// TIA Portal V20 export
DATA_BLOCK "HmiInterface"   // DB204
// stored: Access Published, MemoryReserve 100, Namespace Unit1
   VAR
      AutoStartEnable { ExternalWritable := 'False'} : Bool;
      InitializeEnable { ExternalWritable := 'False'} : Bool;
      camDataBk : Array[1..41] of "LER_typeSoftCamInterface";
   END_VAR
   VAR RETAIN
      BA010 : "LER_typeCommunicationInterface";
      BA015 : "LER_typeCommunicationInterface";
   END_VAR
   VAR
      BA060 { S7_SetPoint := 'True'} : "LER_typeCommunicationInterface";
      BA040 { S7_SetPoint := 'True'} : "LER_typeCommunicationInterface";
      cmFFU { S7_SetPoint := 'True'} : "LER_typeLIU117Interface";
      allBrakeTest : "LER_typeBrakeTestUnitInterface";
      cmPowerMeter_PAC3220 { S7_SetPoint := 'True'} : "LER_typePAC3220Interface";
      cmHandyQRreadDM8700 { S7_SetPoint := 'True'} : "LER_typeDM8700Interface";
      DriveDiagConfig : Struct
         driveObjects : Array[0..41] of "LAF_typeDriveDiagConfig";
         torqueLoad : Array[0.._.LAF_DRV_DIAG_NO_DO] of "LER_typeServoTorqueCalConfigruation";
      END_STRUCT;
      DriveDiagInterfaceHmi : Struct
         diagStatus : "LAF_typeDriveDiagInterfaceHmi";
         torqueLoad { S7_SetPoint := 'True'} : Array[0.._.LAF_DRV_DIAG_NO_DO] of "LER_typeServoTorqueCalInterface";
      END_STRUCT;
      ProductData_DriveSub : Int;
   END_VAR
BEGIN
   // camDataBk[3] : cmCompensatorAxisX
   // camDataBk[4] : cmSepaFeedingRollerAxisB
   // camDataBk[5] : anodeMainPnP1AxisX
   // camDataBk[6] : anodeMainPnP2AxisX
   // camDataBk[7] : cathodeMainPnP1AxisX
   // camDataBk[8] : cathodeMainPnP2AxisX
   // camDataBk[9] : cathodeMainPnP1AxisY
   // camDataBk[10] : cathodeMainPnP1AxisZ
   // camDataBk[11] : anodeMainPnP1AxisY
   // camDataBk[12] : anodeMainPnP1AxisZ
   // camDataBk[13] : cathodeMainPnP2AxisZ
   // camDataBk[14] : anodeMainPnP2AxisZ
   // camDataBk[15] : anodeAlignTableAxisX
   // camDataBk[16] : anodeAlignTableAxisY1
   // camDataBk[17] : anodeAlignTableAxisY2
   // camDataBk[18] : cathodeAlignTableAxisU
   // camDataBk[19] : cathodeAlignTableAxisV
   // camDataBk[20] : cathodeAlignTableAxisW
   // camDataBk[21] : FinalRollerFrontAxisX
   // camDataBk[22] : FinalRollerRearAxisX
   // camDataBk[23] : mendrelAnodeFrontAxisY
   // camDataBk[24] : mendrelAnodeFrontAxisZ
   // camDataBk[25] : mendrelAnodeRearAxisY
   // camDataBk[26] : mendrelAnodeRearAxisZ
   // camDataBk[27] : mendrelCathodeFrontAxisY
   // camDataBk[28] : mendrelCathodeFrontAxisZ
   // camDataBk[29] : mendrelCathodeRearAxisY
   // camDataBk[30] : mendrelCathodeRearAxisZ
   // camDataBk[31] : StackTableAxisZ
   // camDataBk[32] : StackTableOutFrontAxisZ
   // camDataBk[33] : StackTableOutRearAxisZ
   // camDataBk[34] : SepaClampnCutterAxisX
   // camDataBk[35] : SepaClampnCutterAxisZ
   // camDataBk[36] : SepaGripperAxisX
   // camDataBk[37] : SepaGripperAxisZ
   // camDataBk[38] : SepaGripperAxisC
   // camDataBk[39] : JRWinderFrontAxisY
   // camDataBk[40] : JRWinderRearAxisY
   // camDataBk[41] : JRWinderAxisB
   camDataBk[1..4].TargetPosition := 0.0;
   camDataBk[5].TargetPosition := -5.0;
   camDataBk[6].TargetPosition := 546.5;
   camDataBk[7..9].TargetPosition := 0.0;
   camDataBk[10].TargetPosition := 26.2;
   camDataBk[11..12].TargetPosition := 0.0;
   camDataBk[13].TargetPosition := 4.0;
   camDataBk[14].TargetPosition := 3.0;
   camDataBk[15].TargetPosition := -2.08;
   camDataBk[16].TargetPosition := 0.0;
   camDataBk[17].TargetPosition := 8.5;
   camDataBk[18..22].TargetPosition := 0.0;
   camDataBk[23].TargetPosition := 87.68;
   camDataBk[24].TargetPosition := 13.6;
   camDataBk[25].TargetPosition := 8.54;
   camDataBk[26].TargetPosition := -0.1;
   camDataBk[27].TargetPosition := 10.05;
   camDataBk[28].TargetPosition := -0.2;
   camDataBk[29].TargetPosition := 12.45;
   camDataBk[30].TargetPosition := -0.6;
   camDataBk[31].TargetPosition := -20.2;
   camDataBk[32..35].TargetPosition := 0.0;
   camDataBk[36].TargetPosition := 27.5;
   camDataBk[37..38].TargetPosition := 0.0;
   camDataBk[39].TargetPosition := -22.0;
   camDataBk[40..41].TargetPosition := 0.0;
   camDataBk[1..3].ActualPosition := 0.0;
   camDataBk[4].ActualPosition := 70.013;
   camDataBk[5].ActualPosition := 539.942;
   camDataBk[6].ActualPosition := 546.453;
   camDataBk[7].ActualPosition := 0.048;
   camDataBk[8].ActualPosition := -11.987;
   camDataBk[9].ActualPosition := 0.0;
   camDataBk[10].ActualPosition := 4.235;
   camDataBk[11].ActualPosition := 0.0;
   camDataBk[12].ActualPosition := 5.435;
   camDataBk[13].ActualPosition := 4.649;
   camDataBk[14].ActualPosition := 3.012;
   camDataBk[15].ActualPosition := -2.08;
   camDataBk[16].ActualPosition := 0.6;
   camDataBk[17].ActualPosition := 0.0;
   camDataBk[18].ActualPosition := -0.929;
   camDataBk[19].ActualPosition := 0.15;
   camDataBk[20].ActualPosition := -0.959;
   camDataBk[21].ActualPosition := 31.141;
   camDataBk[22].ActualPosition := 0.0;
   camDataBk[23].ActualPosition := -25.432;
   camDataBk[24].ActualPosition := 20.924;
   camDataBk[25].ActualPosition := 8.538;
   camDataBk[26].ActualPosition := 13.346;
   camDataBk[27].ActualPosition := 10.959;
   camDataBk[28].ActualPosition := 2.036;
   camDataBk[29].ActualPosition := 12.418;
   camDataBk[30].ActualPosition := 13.294;
   camDataBk[31].ActualPosition := -20.2;
   camDataBk[32].ActualPosition := -13.254;
   camDataBk[33].ActualPosition := 0.0;
   camDataBk[34].ActualPosition := 245.002;
   camDataBk[35].ActualPosition := 144.852;
   camDataBk[36].ActualPosition := 27.536;
   camDataBk[37].ActualPosition := 158.76;
   camDataBk[38].ActualPosition := -6.304;
   camDataBk[39].ActualPosition := -21.985;
   camDataBk[40].ActualPosition := -17.994;
   camDataBk[41].ActualPosition := 0.34;
   camDataBk[1..41].error := FALSE;
   camDataBk[1..41].status := 16#0000;
   camDataBk[1].position[0..8].SetValue.Negative := 0.0;
   camDataBk[2].position[0..8].SetValue.Negative := 0.0;
   camDataBk[3].position[0..8].SetValue.Negative := 1.0;
   camDataBk[4].position[0].SetValue.Negative := 0.0;
   camDataBk[4].position[1..2].SetValue.Negative := 1.0;
   camDataBk[4].position[3..8].SetValue.Negative := 0.0;
   camDataBk[5].position[0..8].SetValue.Negative := 1.0;
   camDataBk[6].position[0..8].SetValue.Negative := 1.0;
   camDataBk[7].position[0..8].SetValue.Negative := 1.0;
   camDataBk[8].position[0..8].SetValue.Negative := 1.0;
   camDataBk[9].position[0..8].SetValue.Negative := 1.0;
   camDataBk[10].position[0..8].SetValue.Negative := 1.0;
   camDataBk[11].position[0..8].SetValue.Negative := 1.0;
   camDataBk[12].position[0..8].SetValue.Negative := 1.0;
   camDataBk[13].position[0..8].SetValue.Negative := 1.0;
   camDataBk[14].position[0..8].SetValue.Negative := 1.0;
   camDataBk[15].position[0..8].SetValue.Negative := 1.0;
   camDataBk[16].position[0..8].SetValue.Negative := 1.0;
   camDataBk[17].position[0..8].SetValue.Negative := 1.0;
   camDataBk[18].position[0..8].SetValue.Negative := 1.0;
   camDataBk[19].position[0..8].SetValue.Negative := 1.0;
   camDataBk[20].position[0..8].SetValue.Negative := 1.0;
   camDataBk[21].position[0..8].SetValue.Negative := 1.0;
   camDataBk[22].position[0..8].SetValue.Negative := 1.0;
   camDataBk[23].position[0..8].SetValue.Negative := 1.0;
   camDataBk[24].position[0..8].SetValue.Negative := 1.0;
   camDataBk[25].position[0..8].SetValue.Negative := 1.0;
   camDataBk[26].position[0..8].SetValue.Negative := 1.0;
   camDataBk[27].position[0..8].SetValue.Negative := 1.0;
   camDataBk[28].position[0..8].SetValue.Negative := 1.0;
   camDataBk[29].position[0..8].SetValue.Negative := 1.0;
   camDataBk[30].position[0..8].SetValue.Negative := 1.0;
   camDataBk[31].position[0..8].SetValue.Negative := 1.0;
   camDataBk[32].position[0..8].SetValue.Negative := 1.0;
   camDataBk[33].position[0..8].SetValue.Negative := 1.0;
   camDataBk[34].position[0..8].SetValue.Negative := 1.0;
   camDataBk[35].position[0..8].SetValue.Negative := 1.0;
   camDataBk[36].position[0..8].SetValue.Negative := 1.0;
   camDataBk[37].position[0..8].SetValue.Negative := 1.0;
   camDataBk[38].position[0..8].SetValue.Negative := 1.0;
   camDataBk[39].position[0..8].SetValue.Negative := 1.0;
   camDataBk[40].position[0..8].SetValue.Negative := 1.0;
   camDataBk[41].position[0..8].SetValue.Negative := 1.0;
   camDataBk[1].position[0..8].SetValue.Postive := 0.0;
   camDataBk[2].position[0..8].SetValue.Postive := 0.0;
   camDataBk[3].position[0..8].SetValue.Postive := 1.0;
   camDataBk[4].position[0].SetValue.Postive := 0.0;
   camDataBk[4].position[1..2].SetValue.Postive := 1.0;
   camDataBk[4].position[3..8].SetValue.Postive := 0.0;
   camDataBk[5].position[0..8].SetValue.Postive := 1.0;
   camDataBk[6].position[0..8].SetValue.Postive := 1.0;
   camDataBk[7].position[0..5].SetValue.Postive := 1.0;
   camDataBk[7].position[6].SetValue.Postive := 0.001;
   camDataBk[7].position[7..8].SetValue.Postive := 1.0;
   camDataBk[8].position[0..8].SetValue.Postive := 1.0;
   camDataBk[9].position[0..8].SetValue.Postive := 1.0;
   camDataBk[10].position[0..8].SetValue.Postive := 1.0;
   camDataBk[11].position[0..8].SetValue.Postive := 1.0;
   camDataBk[12].position[0..8].SetValue.Postive := 1.0;
   camDataBk[13].position[0..8].SetValue.Postive := 1.0;
   camDataBk[14].position[0..8].SetValue.Postive := 1.0;
   camDataBk[15].position[0..8].SetValue.Postive := 1.0;
   camDataBk[16].position[0..8].SetValue.Postive := 1.0;
   camDataBk[17].position[0..8].SetValue.Postive := 1.0;
   camDataBk[18].position[0..8].SetValue.Postive := 1.0;
   camDataBk[19].position[0..8].SetValue.Postive := 1.0;
   camDataBk[20].position[0..8].SetValue.Postive := 1.0;
   camDataBk[21].position[0..8].SetValue.Postive := 1.0;
   camDataBk[22].position[0..8].SetValue.Postive := 1.0;
   camDataBk[23].position[0..8].SetValue.Postive := 1.0;
   camDataBk[24].position[0..8].SetValue.Postive := 1.0;
   camDataBk[25].position[0..8].SetValue.Postive := 1.0;
   camDataBk[26].position[0..8].SetValue.Postive := 1.0;
   camDataBk[27].position[0..8].SetValue.Postive := 1.0;
   camDataBk[28].position[0..8].SetValue.Postive := 1.0;
   camDataBk[29].position[0..8].SetValue.Postive := 1.0;
   camDataBk[30].position[0..8].SetValue.Postive := 1.0;
   camDataBk[31].position[0..8].SetValue.Postive := 1.0;
   camDataBk[32].position[0..8].SetValue.Postive := 1.0;
   camDataBk[33].position[0..8].SetValue.Postive := 1.0;
   camDataBk[34].position[0..8].SetValue.Postive := 1.0;
   camDataBk[35].position[0..8].SetValue.Postive := 1.0;
   camDataBk[36].position[0..8].SetValue.Postive := 1.0;
   camDataBk[37].position[0..8].SetValue.Postive := 1.0;
   camDataBk[38].position[0..8].SetValue.Postive := 1.0;
   camDataBk[39].position[0..8].SetValue.Postive := 1.0;
   camDataBk[40].position[0..8].SetValue.Postive := 1.0;
   camDataBk[41].position[0..8].SetValue.Postive := 1.0;
   camDataBk[1].position[0..8].ProcessValue.Postive := 0.0;
   camDataBk[2].position[0..8].ProcessValue.Postive := 0.0;
   camDataBk[3].position[0..8].ProcessValue.Postive := 0.0;
   camDataBk[4].position[0].ProcessValue.Postive := 0.0;
   camDataBk[4].position[1..2].ProcessValue.Postive := 1.0;
   camDataBk[4].position[3..8].ProcessValue.Postive := 0.0;
   camDataBk[5].position[0..8].ProcessValue.Postive := 1.0;
   camDataBk[6].position[0..8].ProcessValue.Postive := 1.0;
   camDataBk[7].position[0..5].ProcessValue.Postive := 1.0;
   camDataBk[7].position[6].ProcessValue.Postive := 0.001;
   camDataBk[7].position[7..8].ProcessValue.Postive := 1.0;
   camDataBk[8].position[0..8].ProcessValue.Postive := 1.0;
   camDataBk[9].position[0..8].ProcessValue.Postive := 1.0;
   camDataBk[10].position[0..8].ProcessValue.Postive := 1.0;
   camDataBk[11].position[0..8].ProcessValue.Postive := 1.0;
   camDataBk[12].position[0..8].ProcessValue.Postive := 1.0;
   camDataBk[13].position[0..8].ProcessValue.Postive := 1.0;
   camDataBk[14].position[0..8].ProcessValue.Postive := 1.0;
   camDataBk[15].position[0..8].ProcessValue.Postive := 1.0;
   camDataBk[16].position[0..8].ProcessValue.Postive := 1.0;
   camDataBk[17].position[0..8].ProcessValue.Postive := 1.0;
   camDataBk[18].position[0..8].ProcessValue.Postive := 1.0;
   camDataBk[19].position[0..8].ProcessValue.Postive := 1.0;
   camDataBk[20].position[0..8].ProcessValue.Postive := 1.0;
   camDataBk[21].position[0..8].ProcessValue.Postive := 1.0;
   camDataBk[22].position[0..8].ProcessValue.Postive := 0.0;
   camDataBk[23].position[0..8].ProcessValue.Postive := 1.0;
   camDataBk[24].position[0..8].ProcessValue.Postive := 1.0;
   camDataBk[25].position[0..8].ProcessValue.Postive := 1.0;
   camDataBk[26].position[0..8].ProcessValue.Postive := 1.0;
   camDataBk[27].position[0..8].ProcessValue.Postive := 1.0;
   camDataBk[28].position[0..8].ProcessValue.Postive := 1.0;
   camDataBk[29].position[0..8].ProcessValue.Postive := 1.0;
   camDataBk[30].position[0..8].ProcessValue.Postive := 1.0;
   camDataBk[31].position[0..8].ProcessValue.Postive := 1.0;
   camDataBk[32].position[0..8].ProcessValue.Postive := 1.0;
   camDataBk[33].position[0..8].ProcessValue.Postive := 0.0;
   camDataBk[34].position[0..8].ProcessValue.Postive := 1.0;
   camDataBk[35].position[0..8].ProcessValue.Postive := 1.0;
   camDataBk[36].position[0..8].ProcessValue.Postive := 1.0;
   camDataBk[37].position[0..8].ProcessValue.Postive := 1.0;
   camDataBk[38].position[0..8].ProcessValue.Postive := 1.0;
   camDataBk[39].position[0..8].ProcessValue.Postive := 1.0;
   camDataBk[40].position[0..8].ProcessValue.Postive := 1.0;
   camDataBk[41].position[0..8].ProcessValue.Postive := 1.0;
   camDataBk[1].position[0..8].ProcessValue.Negative := 0.0;
   camDataBk[2].position[0..8].ProcessValue.Negative := 0.0;
   camDataBk[3].position[0..8].ProcessValue.Negative := 0.0;
   camDataBk[4].position[0].ProcessValue.Negative := 0.0;
   camDataBk[4].position[1..2].ProcessValue.Negative := 1.0;
   camDataBk[4].position[3..8].ProcessValue.Negative := 0.0;
   camDataBk[5].position[0..8].ProcessValue.Negative := 1.0;
   camDataBk[6].position[0..8].ProcessValue.Negative := 1.0;
   camDataBk[7].position[0..8].ProcessValue.Negative := 1.0;
   camDataBk[8].position[0..8].ProcessValue.Negative := 1.0;
   camDataBk[9].position[0..8].ProcessValue.Negative := 1.0;
   camDataBk[10].position[0..8].ProcessValue.Negative := 1.0;
   camDataBk[11].position[0..8].ProcessValue.Negative := 1.0;
   camDataBk[12].position[0..8].ProcessValue.Negative := 1.0;
   camDataBk[13].position[0..8].ProcessValue.Negative := 1.0;
   camDataBk[14].position[0..8].ProcessValue.Negative := 1.0;
   camDataBk[15].position[0..8].ProcessValue.Negative := 1.0;
   camDataBk[16].position[0..8].ProcessValue.Negative := 1.0;
   camDataBk[17].position[0..8].ProcessValue.Negative := 1.0;
   camDataBk[18].position[0..8].ProcessValue.Negative := 1.0;
   camDataBk[19].position[0..8].ProcessValue.Negative := 1.0;
   camDataBk[20].position[0..8].ProcessValue.Negative := 1.0;
   camDataBk[21].position[0..8].ProcessValue.Negative := 1.0;
   camDataBk[22].position[0..8].ProcessValue.Negative := 0.0;
   camDataBk[23].position[0..8].ProcessValue.Negative := 1.0;
   camDataBk[24].position[0..8].ProcessValue.Negative := 1.0;
   camDataBk[25].position[0..8].ProcessValue.Negative := 1.0;
   camDataBk[26].position[0..8].ProcessValue.Negative := 1.0;
   camDataBk[27].position[0..8].ProcessValue.Negative := 1.0;
   camDataBk[28].position[0..8].ProcessValue.Negative := 1.0;
   camDataBk[29].position[0..8].ProcessValue.Negative := 1.0;
   camDataBk[30].position[0..8].ProcessValue.Negative := 1.0;
   camDataBk[31].position[0..8].ProcessValue.Negative := 1.0;
   camDataBk[32].position[0..8].ProcessValue.Negative := 1.0;
   camDataBk[33].position[0..8].ProcessValue.Negative := 0.0;
   camDataBk[34].position[0..8].ProcessValue.Negative := 1.0;
   camDataBk[35].position[0..8].ProcessValue.Negative := 1.0;
   camDataBk[36].position[0..8].ProcessValue.Negative := 1.0;
   camDataBk[37].position[0..8].ProcessValue.Negative := 1.0;
   camDataBk[38].position[0..8].ProcessValue.Negative := 1.0;
   camDataBk[39].position[0..8].ProcessValue.Negative := 1.0;
   camDataBk[40].position[0..8].ProcessValue.Negative := 1.0;
   camDataBk[41].position[0..8].ProcessValue.Negative := 1.0;
   camDataBk[1].position[0..8].ProcessValue.SetPos := 0.0;
   camDataBk[2].position[0..8].ProcessValue.SetPos := 0.0;
   camDataBk[3].position[0..8].ProcessValue.SetPos := 0.0;
   camDataBk[4].position[0].ProcessValue.SetPos := 0.0;
   camDataBk[4].position[1].ProcessValue.SetPos := 50.0;
   camDataBk[4].position[2].ProcessValue.SetPos := 70.0;
   camDataBk[4].position[3..8].ProcessValue.SetPos := 0.0;
   camDataBk[5].position[0].ProcessValue.SetPos := 0.0;
   camDataBk[5].position[1].ProcessValue.SetPos := 540.0;
   camDataBk[5].position[2].ProcessValue.SetPos := -5.0;
   camDataBk[5].position[3..8].ProcessValue.SetPos := 0.0;
   camDataBk[6].position[0].ProcessValue.SetPos := 0.0;
   camDataBk[6].position[1].ProcessValue.SetPos := 546.5;
   camDataBk[6].position[2].ProcessValue.SetPos := -3.5;
   camDataBk[6].position[3..8].ProcessValue.SetPos := 0.0;
   camDataBk[7].position[0..1].ProcessValue.SetPos := 0.0;
   camDataBk[7].position[2].ProcessValue.SetPos := 544.0;
   camDataBk[7].position[3..8].ProcessValue.SetPos := 0.0;
   camDataBk[8].position[0].ProcessValue.SetPos := 0.0;
   camDataBk[8].position[1].ProcessValue.SetPos := -12.0;
   camDataBk[8].position[2].ProcessValue.SetPos := 538.0;
   camDataBk[8].position[3..8].ProcessValue.SetPos := 0.0;
   camDataBk[9].position[0..8].ProcessValue.SetPos := 0.0;
   camDataBk[10].position[0].ProcessValue.SetPos := 0.0;
   camDataBk[10].position[1].ProcessValue.SetPos := 0.3;
   camDataBk[10].position[2].ProcessValue.SetPos := 26.2;
   camDataBk[10].position[3..8].ProcessValue.SetPos := 0.0;
   camDataBk[11].position[0..8].ProcessValue.SetPos := 0.0;
   camDataBk[12].position[0..1].ProcessValue.SetPos := 4.0;
   camDataBk[12].position[2].ProcessValue.SetPos := 23.0;
   camDataBk[12].position[3].ProcessValue.SetPos := 26.3;
   camDataBk[12].position[4..8].ProcessValue.SetPos := 0.0;
   camDataBk[13].position[0].ProcessValue.SetPos := 0.0;
   camDataBk[13].position[1].ProcessValue.SetPos := 4.0;
   camDataBk[13].position[2].ProcessValue.SetPos := 26.6;
   camDataBk[13].position[3..8].ProcessValue.SetPos := 0.0;
   camDataBk[14].position[0].ProcessValue.SetPos := 0.0;
   camDataBk[14].position[1].ProcessValue.SetPos := 3.0;
   camDataBk[14].position[2].ProcessValue.SetPos := 25.5;
   camDataBk[14].position[3].ProcessValue.SetPos := 26.5;
   camDataBk[14].position[4..8].ProcessValue.SetPos := 0.0;
   camDataBk[15].position[0].ProcessValue.SetPos := 0.0;
   camDataBk[15].position[1].ProcessValue.SetPos := -2.08;
   camDataBk[15].position[2..3].ProcessValue.SetPos := -4.08;
   camDataBk[15].position[4].ProcessValue.SetPos := -2.08;
   camDataBk[15].position[5..7].ProcessValue.SetPos := -0.08;
   camDataBk[15].position[8].ProcessValue.SetPos := 6.42;
   camDataBk[16].position[0].ProcessValue.SetPos := 0.0;
   camDataBk[16].position[1..2].ProcessValue.SetPos := 0.6;
   camDataBk[16].position[3..5].ProcessValue.SetPos := 2.6;
   camDataBk[16].position[6].ProcessValue.SetPos := 0.6;
   camDataBk[16].position[7].ProcessValue.SetPos := -1.4;
   camDataBk[16].position[8].ProcessValue.SetPos := 9.1;
   camDataBk[17].position[0..7].ProcessValue.SetPos := 0.0;
   camDataBk[17].position[8].ProcessValue.SetPos := 8.5;
   camDataBk[18].position[0].ProcessValue.SetPos := 0.0;
   camDataBk[18].position[1].ProcessValue.SetPos := -0.93;
   camDataBk[18].position[2..3].ProcessValue.SetPos := 1.07;
   camDataBk[18].position[4].ProcessValue.SetPos := -0.93;
   camDataBk[18].position[5..7].ProcessValue.SetPos := -2.93;
   camDataBk[18].position[8].ProcessValue.SetPos := -0.93;
   camDataBk[19].position[0].ProcessValue.SetPos := 0.0;
   camDataBk[19].position[1..2].ProcessValue.SetPos := 0.15;
   camDataBk[19].position[3..5].ProcessValue.SetPos := 2.15;
   camDataBk[19].position[6].ProcessValue.SetPos := 0.15;
   camDataBk[19].position[7].ProcessValue.SetPos := -1.85;
   camDataBk[19].position[8].ProcessValue.SetPos := 0.15;
   camDataBk[20].position[0].ProcessValue.SetPos := 0.0;
   camDataBk[20].position[1..2].ProcessValue.SetPos := -0.96;
   camDataBk[20].position[3..5].ProcessValue.SetPos := -2.96;
   camDataBk[20].position[6].ProcessValue.SetPos := -0.96;
   camDataBk[20].position[7].ProcessValue.SetPos := 1.04;
   camDataBk[20].position[8].ProcessValue.SetPos := -0.96;
   camDataBk[21].position[0].ProcessValue.SetPos := 0.0;
   camDataBk[21].position[1].ProcessValue.SetPos := -1.0;
   camDataBk[21].position[2].ProcessValue.SetPos := 345.0;
   camDataBk[21].position[3..8].ProcessValue.SetPos := 0.0;
   camDataBk[22].position[0..8].ProcessValue.SetPos := 0.0;
   camDataBk[23].position[0].ProcessValue.SetPos := 0.0;
   camDataBk[23].position[1].ProcessValue.SetPos := 12.44;
   camDataBk[23].position[2].ProcessValue.SetPos := 87.68;
   camDataBk[23].position[3..8].ProcessValue.SetPos := 0.0;
   camDataBk[24].position[0].ProcessValue.SetPos := 0.0;
   camDataBk[24].position[1].ProcessValue.SetPos := -2.8;
   camDataBk[24].position[2].ProcessValue.SetPos := 13.6;
   camDataBk[24].position[3..8].ProcessValue.SetPos := 0.0;
   camDataBk[25].position[0].ProcessValue.SetPos := 0.0;
   camDataBk[25].position[1].ProcessValue.SetPos := 8.54;
   camDataBk[25].position[2].ProcessValue.SetPos := 84.03;
   camDataBk[25].position[3..8].ProcessValue.SetPos := 0.0;
   camDataBk[26].position[0].ProcessValue.SetPos := 0.0;
   camDataBk[26].position[1].ProcessValue.SetPos := -0.1;
   camDataBk[26].position[2].ProcessValue.SetPos := 15.7;
   camDataBk[26].position[3..8].ProcessValue.SetPos := 0.0;
   camDataBk[27].position[0].ProcessValue.SetPos := 0.0;
   camDataBk[27].position[1].ProcessValue.SetPos := 10.05;
   camDataBk[27].position[2].ProcessValue.SetPos := 85.43;
   camDataBk[27].position[3..8].ProcessValue.SetPos := 0.0;
   camDataBk[28].position[0].ProcessValue.SetPos := 0.0;
   camDataBk[28].position[1].ProcessValue.SetPos := -0.2;
   camDataBk[28].position[2].ProcessValue.SetPos := 14.4;
   camDataBk[28].position[3..8].ProcessValue.SetPos := 0.0;
   camDataBk[29].position[0].ProcessValue.SetPos := 0.0;
   camDataBk[29].position[1].ProcessValue.SetPos := 12.45;
   camDataBk[29].position[2].ProcessValue.SetPos := 88.92;
   camDataBk[29].position[3..8].ProcessValue.SetPos := 0.0;
   camDataBk[30].position[0].ProcessValue.SetPos := 0.0;
   camDataBk[30].position[1].ProcessValue.SetPos := -0.6;
   camDataBk[30].position[2].ProcessValue.SetPos := 14.6;
   camDataBk[30].position[3..8].ProcessValue.SetPos := 0.0;
   camDataBk[31].position[0].ProcessValue.SetPos := 0.0;
   camDataBk[31].position[1].ProcessValue.SetPos := -20.2;
   camDataBk[31].position[2].ProcessValue.SetPos := 0.0;
   camDataBk[31].position[3].ProcessValue.SetPos := -3.5;
   camDataBk[31].position[4..8].ProcessValue.SetPos := 0.0;
   camDataBk[32].position[0].ProcessValue.SetPos := 0.0;
   camDataBk[32].position[1].ProcessValue.SetPos := -10.76;
   camDataBk[32].position[2].ProcessValue.SetPos := 174.0;
   camDataBk[32].position[3..8].ProcessValue.SetPos := 0.0;
   camDataBk[33].position[0..8].ProcessValue.SetPos := 0.0;
   camDataBk[34].position[0].ProcessValue.SetPos := 0.0;
   camDataBk[34].position[1].ProcessValue.SetPos := 245.0;
   camDataBk[34].position[2].ProcessValue.SetPos := 48.2;
   camDataBk[34].position[3].ProcessValue.SetPos := 720.0;
   camDataBk[34].position[4..8].ProcessValue.SetPos := 0.0;
   camDataBk[35].position[0].ProcessValue.SetPos := 0.0;
   camDataBk[35].position[1].ProcessValue.SetPos := 141.0;
   camDataBk[35].position[2].ProcessValue.SetPos := 143.8;
   camDataBk[35].position[3].ProcessValue.SetPos := 160.0;
   camDataBk[35].position[4..8].ProcessValue.SetPos := 0.0;
   camDataBk[36].position[0].ProcessValue.SetPos := 0.0;
   camDataBk[36].position[1].ProcessValue.SetPos := 27.5;
   camDataBk[36].position[2..3].ProcessValue.SetPos := 1706.6;
   camDataBk[36].position[4].ProcessValue.SetPos := 245.0;
   camDataBk[36].position[5].ProcessValue.SetPos := 27.5;
   camDataBk[36].position[6].ProcessValue.SetPos := 227.5;
   camDataBk[36].position[7].ProcessValue.SetPos := 0.0;
   camDataBk[36].position[8].ProcessValue.SetPos := 179.3;
   camDataBk[37].position[0].ProcessValue.SetPos := 0.0;
   camDataBk[37].position[1].ProcessValue.SetPos := 233.0;
   camDataBk[37].position[2].ProcessValue.SetPos := 280.6;
   camDataBk[37].position[3].ProcessValue.SetPos := 159.6;
   camDataBk[37].position[4].ProcessValue.SetPos := 18.75;
   camDataBk[37].position[5].ProcessValue.SetPos := 233.5;
   camDataBk[37].position[6].ProcessValue.SetPos := 146.0;
   camDataBk[37].position[7..8].ProcessValue.SetPos := 0.0;
   camDataBk[38].position[0].ProcessValue.SetPos := 0.0;
   camDataBk[38].position[1].ProcessValue.SetPos := -1.43;
   camDataBk[38].position[2].ProcessValue.SetPos := 178.4;
   camDataBk[38].position[3].ProcessValue.SetPos := 88.4;
   camDataBk[38].position[4..8].ProcessValue.SetPos := 0.0;
   camDataBk[39].position[0].ProcessValue.SetPos := 0.0;
   camDataBk[39].position[1].ProcessValue.SetPos := -22.0;
   camDataBk[39].position[2].ProcessValue.SetPos := 160.0;
   camDataBk[39].position[3..8].ProcessValue.SetPos := 0.0;
   camDataBk[40].position[0].ProcessValue.SetPos := 0.0;
   camDataBk[40].position[1..2].ProcessValue.SetPos := -18.0;
   camDataBk[40].position[3..8].ProcessValue.SetPos := 0.0;
   camDataBk[41].position[0..8].ProcessValue.SetPos := 0.0;
   camDataBk[1].position[0..8].ProcessValue.inPos := FALSE;
   camDataBk[2].position[0..8].ProcessValue.inPos := FALSE;
   camDataBk[3].position[0..8].ProcessValue.inPos := FALSE;
   camDataBk[4].position[0..1].ProcessValue.inPos := FALSE;
   camDataBk[4].position[2].ProcessValue.inPos := TRUE;
   camDataBk[4].position[3..8].ProcessValue.inPos := FALSE;
   camDataBk[5].position[0].ProcessValue.inPos := FALSE;
   camDataBk[5].position[1].ProcessValue.inPos := TRUE;
   camDataBk[5].position[2..8].ProcessValue.inPos := FALSE;
   camDataBk[6].position[0].ProcessValue.inPos := FALSE;
   camDataBk[6].position[1].ProcessValue.inPos := TRUE;
   camDataBk[6].position[2..8].ProcessValue.inPos := FALSE;
   camDataBk[7].position[0..1].ProcessValue.inPos := TRUE;
   camDataBk[7].position[2].ProcessValue.inPos := FALSE;
   camDataBk[7].position[3..5].ProcessValue.inPos := TRUE;
   camDataBk[7].position[6].ProcessValue.inPos := FALSE;
   camDataBk[7].position[7..8].ProcessValue.inPos := TRUE;
   camDataBk[8].position[0].ProcessValue.inPos := FALSE;
   camDataBk[8].position[1].ProcessValue.inPos := TRUE;
   camDataBk[8].position[2..8].ProcessValue.inPos := FALSE;
   camDataBk[9].position[0..8].ProcessValue.inPos := TRUE;
   camDataBk[10].position[0..8].ProcessValue.inPos := FALSE;
   camDataBk[11].position[0..8].ProcessValue.inPos := TRUE;
   camDataBk[12].position[0..8].ProcessValue.inPos := FALSE;
   camDataBk[13].position[0].ProcessValue.inPos := FALSE;
   camDataBk[13].position[1].ProcessValue.inPos := TRUE;
   camDataBk[13].position[2..8].ProcessValue.inPos := FALSE;
   camDataBk[14].position[0].ProcessValue.inPos := FALSE;
   camDataBk[14].position[1].ProcessValue.inPos := TRUE;
   camDataBk[14].position[2..8].ProcessValue.inPos := FALSE;
   camDataBk[15].position[0].ProcessValue.inPos := FALSE;
   camDataBk[15].position[1].ProcessValue.inPos := TRUE;
   camDataBk[15].position[2..3].ProcessValue.inPos := FALSE;
   camDataBk[15].position[4].ProcessValue.inPos := TRUE;
   camDataBk[15].position[5..8].ProcessValue.inPos := FALSE;
   camDataBk[16].position[0..2].ProcessValue.inPos := TRUE;
   camDataBk[16].position[3..5].ProcessValue.inPos := FALSE;
   camDataBk[16].position[6].ProcessValue.inPos := TRUE;
   camDataBk[16].position[7..8].ProcessValue.inPos := FALSE;
   camDataBk[17].position[0..7].ProcessValue.inPos := TRUE;
   camDataBk[17].position[8].ProcessValue.inPos := FALSE;
   camDataBk[18].position[0..1].ProcessValue.inPos := TRUE;
   camDataBk[18].position[2..3].ProcessValue.inPos := FALSE;
   camDataBk[18].position[4].ProcessValue.inPos := TRUE;
   camDataBk[18].position[5..7].ProcessValue.inPos := FALSE;
   camDataBk[18].position[8].ProcessValue.inPos := TRUE;
   camDataBk[19].position[0..2].ProcessValue.inPos := TRUE;
   camDataBk[19].position[3..5].ProcessValue.inPos := FALSE;
   camDataBk[19].position[6].ProcessValue.inPos := TRUE;
   camDataBk[19].position[7].ProcessValue.inPos := FALSE;
   camDataBk[19].position[8].ProcessValue.inPos := TRUE;
   camDataBk[20].position[0..2].ProcessValue.inPos := TRUE;
   camDataBk[20].position[3..5].ProcessValue.inPos := FALSE;
   camDataBk[20].position[6].ProcessValue.inPos := TRUE;
   camDataBk[20].position[7].ProcessValue.inPos := FALSE;
   camDataBk[20].position[8].ProcessValue.inPos := TRUE;
   camDataBk[21].position[0..8].ProcessValue.inPos := FALSE;
   camDataBk[22].position[0..8].ProcessValue.inPos := FALSE;
   camDataBk[23].position[0..8].ProcessValue.inPos := FALSE;
   camDataBk[24].position[0..8].ProcessValue.inPos := FALSE;
   camDataBk[25].position[0].ProcessValue.inPos := FALSE;
   camDataBk[25].position[1].ProcessValue.inPos := TRUE;
   camDataBk[25].position[2..8].ProcessValue.inPos := FALSE;
   camDataBk[26].position[0..8].ProcessValue.inPos := FALSE;
   camDataBk[27].position[0].ProcessValue.inPos := FALSE;
   camDataBk[27].position[1].ProcessValue.inPos := TRUE;
   camDataBk[27].position[2..8].ProcessValue.inPos := FALSE;
   camDataBk[28].position[0..8].ProcessValue.inPos := FALSE;
   camDataBk[29].position[0].ProcessValue.inPos := FALSE;
   camDataBk[29].position[1].ProcessValue.inPos := TRUE;
   camDataBk[29].position[2..8].ProcessValue.inPos := FALSE;
   camDataBk[30].position[0..8].ProcessValue.inPos := FALSE;
   camDataBk[31].position[0].ProcessValue.inPos := FALSE;
   camDataBk[31].position[1].ProcessValue.inPos := TRUE;
   camDataBk[31].position[2..8].ProcessValue.inPos := FALSE;
   camDataBk[32].position[0..8].ProcessValue.inPos := FALSE;
   camDataBk[33].position[0..8].ProcessValue.inPos := FALSE;
   camDataBk[34].position[0].ProcessValue.inPos := FALSE;
   camDataBk[34].position[1].ProcessValue.inPos := TRUE;
   camDataBk[34].position[2..8].ProcessValue.inPos := FALSE;
   camDataBk[35].position[0..8].ProcessValue.inPos := FALSE;
   camDataBk[36].position[0].ProcessValue.inPos := FALSE;
   camDataBk[36].position[1].ProcessValue.inPos := TRUE;
   camDataBk[36].position[2..4].ProcessValue.inPos := FALSE;
   camDataBk[36].position[5].ProcessValue.inPos := TRUE;
   camDataBk[36].position[6..8].ProcessValue.inPos := FALSE;
   camDataBk[37].position[0..2].ProcessValue.inPos := FALSE;
   camDataBk[37].position[3].ProcessValue.inPos := TRUE;
   camDataBk[37].position[4..8].ProcessValue.inPos := FALSE;
   camDataBk[38].position[0..8].ProcessValue.inPos := FALSE;
   camDataBk[39].position[0].ProcessValue.inPos := FALSE;
   camDataBk[39].position[1].ProcessValue.inPos := TRUE;
   camDataBk[39].position[2..8].ProcessValue.inPos := FALSE;
   camDataBk[40].position[0].ProcessValue.inPos := FALSE;
   camDataBk[40].position[1..2].ProcessValue.inPos := TRUE;
   camDataBk[40].position[3..8].ProcessValue.inPos := FALSE;
   camDataBk[41].position[0..8].ProcessValue.inPos := TRUE;
   camDataBk[1].position[0..8].ProcessValue.isBefore := FALSE;
   camDataBk[2].position[0..8].ProcessValue.isBefore := FALSE;
   camDataBk[3].position[0..8].ProcessValue.isBefore := FALSE;
   camDataBk[4].position[0..8].ProcessValue.isBefore := FALSE;
   camDataBk[5].position[0..8].ProcessValue.isBefore := FALSE;
   camDataBk[6].position[0..8].ProcessValue.isBefore := FALSE;
   camDataBk[7].position[0..1].ProcessValue.isBefore := FALSE;
   camDataBk[7].position[2].ProcessValue.isBefore := TRUE;
   camDataBk[7].position[3..8].ProcessValue.isBefore := FALSE;
   camDataBk[8].position[0].ProcessValue.isBefore := TRUE;
   camDataBk[8].position[1].ProcessValue.isBefore := FALSE;
   camDataBk[8].position[2..8].ProcessValue.isBefore := TRUE;
   camDataBk[9].position[0..8].ProcessValue.isBefore := FALSE;
   camDataBk[10].position[0..1].ProcessValue.isBefore := FALSE;
   camDataBk[10].position[2].ProcessValue.isBefore := TRUE;
   camDataBk[10].position[3..8].ProcessValue.isBefore := FALSE;
   camDataBk[11].position[0..8].ProcessValue.isBefore := FALSE;
   camDataBk[12].position[0..1].ProcessValue.isBefore := FALSE;
   camDataBk[12].position[2..3].ProcessValue.isBefore := TRUE;
   camDataBk[12].position[4..8].ProcessValue.isBefore := FALSE;
   camDataBk[13].position[0..1].ProcessValue.isBefore := FALSE;
   camDataBk[13].position[2].ProcessValue.isBefore := TRUE;
   camDataBk[13].position[3..8].ProcessValue.isBefore := FALSE;
   camDataBk[14].position[0..1].ProcessValue.isBefore := FALSE;
   camDataBk[14].position[2..3].ProcessValue.isBefore := TRUE;
   camDataBk[14].position[4..8].ProcessValue.isBefore := FALSE;
   camDataBk[15].position[0].ProcessValue.isBefore := TRUE;
   camDataBk[15].position[1..4].ProcessValue.isBefore := FALSE;
   camDataBk[15].position[5..8].ProcessValue.isBefore := TRUE;
   camDataBk[16].position[0..2].ProcessValue.isBefore := FALSE;
   camDataBk[16].position[3..5].ProcessValue.isBefore := TRUE;
   camDataBk[16].position[6..7].ProcessValue.isBefore := FALSE;
   camDataBk[16].position[8].ProcessValue.isBefore := TRUE;
   camDataBk[17].position[0..7].ProcessValue.isBefore := FALSE;
   camDataBk[17].position[8].ProcessValue.isBefore := TRUE;
   camDataBk[18].position[0..1].ProcessValue.isBefore := FALSE;
   camDataBk[18].position[2..3].ProcessValue.isBefore := TRUE;
   camDataBk[18].position[4..8].ProcessValue.isBefore := FALSE;
   camDataBk[19].position[0..2].ProcessValue.isBefore := FALSE;
   camDataBk[19].position[3..5].ProcessValue.isBefore := TRUE;
   camDataBk[19].position[6..8].ProcessValue.isBefore := FALSE;
   camDataBk[20].position[0..6].ProcessValue.isBefore := FALSE;
   camDataBk[20].position[7].ProcessValue.isBefore := TRUE;
   camDataBk[20].position[8].ProcessValue.isBefore := FALSE;
   camDataBk[21].position[0..1].ProcessValue.isBefore := FALSE;
   camDataBk[21].position[2].ProcessValue.isBefore := TRUE;
   camDataBk[21].position[3..8].ProcessValue.isBefore := FALSE;
   camDataBk[22].position[0..8].ProcessValue.isBefore := FALSE;
   camDataBk[23].position[0..8].ProcessValue.isBefore := TRUE;
   camDataBk[24].position[0..8].ProcessValue.isBefore := FALSE;
   camDataBk[25].position[0..1].ProcessValue.isBefore := FALSE;
   camDataBk[25].position[2].ProcessValue.isBefore := TRUE;
   camDataBk[25].position[3..8].ProcessValue.isBefore := FALSE;
   camDataBk[26].position[0..1].ProcessValue.isBefore := FALSE;
   camDataBk[26].position[2].ProcessValue.isBefore := TRUE;
   camDataBk[26].position[3..8].ProcessValue.isBefore := FALSE;
   camDataBk[27].position[0..1].ProcessValue.isBefore := FALSE;
   camDataBk[27].position[2].ProcessValue.isBefore := TRUE;
   camDataBk[27].position[3..8].ProcessValue.isBefore := FALSE;
   camDataBk[28].position[0..1].ProcessValue.isBefore := FALSE;
   camDataBk[28].position[2].ProcessValue.isBefore := TRUE;
   camDataBk[28].position[3..8].ProcessValue.isBefore := FALSE;
   camDataBk[29].position[0..1].ProcessValue.isBefore := FALSE;
   camDataBk[29].position[2].ProcessValue.isBefore := TRUE;
   camDataBk[29].position[3..8].ProcessValue.isBefore := FALSE;
   camDataBk[30].position[0..1].ProcessValue.isBefore := FALSE;
   camDataBk[30].position[2].ProcessValue.isBefore := TRUE;
   camDataBk[30].position[3..8].ProcessValue.isBefore := FALSE;
   camDataBk[31].position[0].ProcessValue.isBefore := TRUE;
   camDataBk[31].position[1].ProcessValue.isBefore := FALSE;
   camDataBk[31].position[2..8].ProcessValue.isBefore := TRUE;
   camDataBk[32].position[0..8].ProcessValue.isBefore := TRUE;
   camDataBk[33].position[0..8].ProcessValue.isBefore := FALSE;
   camDataBk[34].position[0..2].ProcessValue.isBefore := FALSE;
   camDataBk[34].position[3].ProcessValue.isBefore := TRUE;
   camDataBk[34].position[4..8].ProcessValue.isBefore := FALSE;
   camDataBk[35].position[0..2].ProcessValue.isBefore := FALSE;
   camDataBk[35].position[3].ProcessValue.isBefore := TRUE;
   camDataBk[35].position[4..8].ProcessValue.isBefore := FALSE;
   camDataBk[36].position[0..1].ProcessValue.isBefore := FALSE;
   camDataBk[36].position[2..4].ProcessValue.isBefore := TRUE;
   camDataBk[36].position[5].ProcessValue.isBefore := FALSE;
   camDataBk[36].position[6].ProcessValue.isBefore := TRUE;
   camDataBk[36].position[7].ProcessValue.isBefore := FALSE;
   camDataBk[36].position[8].ProcessValue.isBefore := TRUE;
   camDataBk[37].position[0].ProcessValue.isBefore := FALSE;
   camDataBk[37].position[1..2].ProcessValue.isBefore := TRUE;
   camDataBk[37].position[3..4].ProcessValue.isBefore := FALSE;
   camDataBk[37].position[5].ProcessValue.isBefore := TRUE;
   camDataBk[37].position[6..8].ProcessValue.isBefore := FALSE;
   camDataBk[38].position[0..8].ProcessValue.isBefore := TRUE;
   camDataBk[39].position[0].ProcessValue.isBefore := TRUE;
   camDataBk[39].position[1].ProcessValue.isBefore := FALSE;
   camDataBk[39].position[2..8].ProcessValue.isBefore := TRUE;
   camDataBk[40].position[0].ProcessValue.isBefore := TRUE;
   camDataBk[40].position[1..2].ProcessValue.isBefore := FALSE;
   camDataBk[40].position[3..8].ProcessValue.isBefore := TRUE;
   camDataBk[41].position[0..8].ProcessValue.isBefore := FALSE;
   camDataBk[1].position[0..8].ProcessValue.isAfter := FALSE;
   camDataBk[2].position[0..8].ProcessValue.isAfter := FALSE;
   camDataBk[3].position[0..8].ProcessValue.isAfter := FALSE;
   camDataBk[4].position[0..1].ProcessValue.isAfter := TRUE;
   camDataBk[4].position[2].ProcessValue.isAfter := FALSE;
   camDataBk[4].position[3..8].ProcessValue.isAfter := TRUE;
   camDataBk[5].position[0].ProcessValue.isAfter := TRUE;
   camDataBk[5].position[1].ProcessValue.isAfter := FALSE;
   camDataBk[5].position[2..8].ProcessValue.isAfter := TRUE;
   camDataBk[6].position[0].ProcessValue.isAfter := TRUE;
   camDataBk[6].position[1].ProcessValue.isAfter := FALSE;
   camDataBk[6].position[2..8].ProcessValue.isAfter := TRUE;
   camDataBk[7].position[0..5].ProcessValue.isAfter := FALSE;
   camDataBk[7].position[6].ProcessValue.isAfter := TRUE;
   camDataBk[7].position[7..8].ProcessValue.isAfter := FALSE;
   camDataBk[8].position[0..8].ProcessValue.isAfter := FALSE;
   camDataBk[9].position[0..8].ProcessValue.isAfter := FALSE;
   camDataBk[10].position[0..1].ProcessValue.isAfter := TRUE;
   camDataBk[10].position[2].ProcessValue.isAfter := FALSE;
   camDataBk[10].position[3..8].ProcessValue.isAfter := TRUE;
   camDataBk[11].position[0..8].ProcessValue.isAfter := FALSE;
   camDataBk[12].position[0..1].ProcessValue.isAfter := TRUE;
   camDataBk[12].position[2..3].ProcessValue.isAfter := FALSE;
   camDataBk[12].position[4..8].ProcessValue.isAfter := TRUE;
   camDataBk[13].position[0].ProcessValue.isAfter := TRUE;
   camDataBk[13].position[1..2].ProcessValue.isAfter := FALSE;
   camDataBk[13].position[3..8].ProcessValue.isAfter := TRUE;
   camDataBk[14].position[0].ProcessValue.isAfter := TRUE;
   camDataBk[14].position[1..3].ProcessValue.isAfter := FALSE;
   camDataBk[14].position[4..8].ProcessValue.isAfter := TRUE;
   camDataBk[15].position[0..1].ProcessValue.isAfter := FALSE;
   camDataBk[15].position[2..3].ProcessValue.isAfter := TRUE;
   camDataBk[15].position[4..8].ProcessValue.isAfter := FALSE;
   camDataBk[16].position[0..6].ProcessValue.isAfter := FALSE;
   camDataBk[16].position[7].ProcessValue.isAfter := TRUE;
   camDataBk[16].position[8].ProcessValue.isAfter := FALSE;
   camDataBk[17].position[0..8].ProcessValue.isAfter := FALSE;
   camDataBk[18].position[0..4].ProcessValue.isAfter := FALSE;
   camDataBk[18].position[5..7].ProcessValue.isAfter := TRUE;
   camDataBk[18].position[8].ProcessValue.isAfter := FALSE;
   camDataBk[19].position[0..6].ProcessValue.isAfter := FALSE;
   camDataBk[19].position[7].ProcessValue.isAfter := TRUE;
   camDataBk[19].position[8].ProcessValue.isAfter := FALSE;
   camDataBk[20].position[0..2].ProcessValue.isAfter := FALSE;
   camDataBk[20].position[3..5].ProcessValue.isAfter := TRUE;
   camDataBk[20].position[6..8].ProcessValue.isAfter := FALSE;
   camDataBk[21].position[0..1].ProcessValue.isAfter := TRUE;
   camDataBk[21].position[2].ProcessValue.isAfter := FALSE;
   camDataBk[21].position[3..8].ProcessValue.isAfter := TRUE;
   camDataBk[22].position[0..8].ProcessValue.isAfter := FALSE;
   camDataBk[23].position[0..8].ProcessValue.isAfter := FALSE;
   camDataBk[24].position[0..8].ProcessValue.isAfter := TRUE;
   camDataBk[25].position[0].ProcessValue.isAfter := TRUE;
   camDataBk[25].position[1..2].ProcessValue.isAfter := FALSE;
   camDataBk[25].position[3..8].ProcessValue.isAfter := TRUE;
   camDataBk[26].position[0..1].ProcessValue.isAfter := TRUE;
   camDataBk[26].position[2].ProcessValue.isAfter := FALSE;
   camDataBk[26].position[3..8].ProcessValue.isAfter := TRUE;
   camDataBk[27].position[0].ProcessValue.isAfter := TRUE;
   camDataBk[27].position[1..2].ProcessValue.isAfter := FALSE;
   camDataBk[27].position[3..8].ProcessValue.isAfter := TRUE;
   camDataBk[28].position[0..1].ProcessValue.isAfter := TRUE;
   camDataBk[28].position[2].ProcessValue.isAfter := FALSE;
   camDataBk[28].position[3..8].ProcessValue.isAfter := TRUE;
   camDataBk[29].position[0].ProcessValue.isAfter := TRUE;
   camDataBk[29].position[1..2].ProcessValue.isAfter := FALSE;
   camDataBk[29].position[3..8].ProcessValue.isAfter := TRUE;
   camDataBk[30].position[0..1].ProcessValue.isAfter := TRUE;
   camDataBk[30].position[2].ProcessValue.isAfter := FALSE;
   camDataBk[30].position[3..8].ProcessValue.isAfter := TRUE;
   camDataBk[31].position[0..8].ProcessValue.isAfter := FALSE;
   camDataBk[32].position[0..8].ProcessValue.isAfter := FALSE;
   camDataBk[33].position[0..8].ProcessValue.isAfter := FALSE;
   camDataBk[34].position[0].ProcessValue.isAfter := TRUE;
   camDataBk[34].position[1].ProcessValue.isAfter := FALSE;
   camDataBk[34].position[2].ProcessValue.isAfter := TRUE;
   camDataBk[34].position[3].ProcessValue.isAfter := FALSE;
   camDataBk[34].position[4..8].ProcessValue.isAfter := TRUE;
   camDataBk[35].position[0..2].ProcessValue.isAfter := TRUE;
   camDataBk[35].position[3].ProcessValue.isAfter := FALSE;
   camDataBk[35].position[4..8].ProcessValue.isAfter := TRUE;
   camDataBk[36].position[0].ProcessValue.isAfter := TRUE;
   camDataBk[36].position[1..6].ProcessValue.isAfter := FALSE;
   camDataBk[36].position[7].ProcessValue.isAfter := TRUE;
   camDataBk[36].position[8].ProcessValue.isAfter := FALSE;
   camDataBk[37].position[0].ProcessValue.isAfter := TRUE;
   camDataBk[37].position[1..3].ProcessValue.isAfter := FALSE;
   camDataBk[37].position[4].ProcessValue.isAfter := TRUE;
   camDataBk[37].position[5].ProcessValue.isAfter := FALSE;
   camDataBk[37].position[6..8].ProcessValue.isAfter := TRUE;
   camDataBk[38].position[0..8].ProcessValue.isAfter := FALSE;
   camDataBk[39].position[0..8].ProcessValue.isAfter := FALSE;
   camDataBk[40].position[0..8].ProcessValue.isAfter := FALSE;
   camDataBk[41].position[0..8].ProcessValue.isAfter := FALSE;
   camDataBk[1].position[0..8].ProcessValue.PosName := WSTRING#'';
   camDataBk[2].position[0..8].ProcessValue.PosName := WSTRING#'';
   camDataBk[3].position[0..8].ProcessValue.PosName := WSTRING#'';
   camDataBk[4].position[0..8].ProcessValue.PosName := WSTRING#'';
   camDataBk[5].position[0..8].ProcessValue.PosName := WSTRING#'';
   camDataBk[6].position[0..8].ProcessValue.PosName := WSTRING#'';
   camDataBk[7].position[0..8].ProcessValue.PosName := WSTRING#'';
   camDataBk[8].position[0..8].ProcessValue.PosName := WSTRING#'';
   camDataBk[9].position[0..8].ProcessValue.PosName := WSTRING#'';
   camDataBk[10].position[0..8].ProcessValue.PosName := WSTRING#'';
   camDataBk[11].position[0..8].ProcessValue.PosName := WSTRING#'';
   camDataBk[12].position[0..8].ProcessValue.PosName := WSTRING#'';
   camDataBk[13].position[0..8].ProcessValue.PosName := WSTRING#'';
   camDataBk[14].position[0..8].ProcessValue.PosName := WSTRING#'';
   camDataBk[15].position[0..8].ProcessValue.PosName := WSTRING#'';
   camDataBk[16].position[0..8].ProcessValue.PosName := WSTRING#'';
   camDataBk[17].position[0..8].ProcessValue.PosName := WSTRING#'';
   camDataBk[18].position[0..8].ProcessValue.PosName := WSTRING#'';
   camDataBk[19].position[0..8].ProcessValue.PosName := WSTRING#'';
   camDataBk[20].position[0..8].ProcessValue.PosName := WSTRING#'';
   camDataBk[21].position[0..8].ProcessValue.PosName := WSTRING#'';
   camDataBk[22].position[0..8].ProcessValue.PosName := WSTRING#'';
   camDataBk[23].position[0..8].ProcessValue.PosName := WSTRING#'';
   camDataBk[24].position[0..8].ProcessValue.PosName := WSTRING#'';
   camDataBk[25].position[0..8].ProcessValue.PosName := WSTRING#'';
   camDataBk[26].position[0..8].ProcessValue.PosName := WSTRING#'';
   camDataBk[27].position[0..8].ProcessValue.PosName := WSTRING#'';
   camDataBk[28].position[0..8].ProcessValue.PosName := WSTRING#'';
   camDataBk[29].position[0..8].ProcessValue.PosName := WSTRING#'';
   camDataBk[30].position[0..8].ProcessValue.PosName := WSTRING#'';
   camDataBk[31].position[0..8].ProcessValue.PosName := WSTRING#'';
   camDataBk[32].position[0..8].ProcessValue.PosName := WSTRING#'';
   camDataBk[33].position[0..8].ProcessValue.PosName := WSTRING#'';
   camDataBk[34].position[0..8].ProcessValue.PosName := WSTRING#'';
   camDataBk[35].position[0..8].ProcessValue.PosName := WSTRING#'';
   camDataBk[36].position[0..8].ProcessValue.PosName := WSTRING#'';
   camDataBk[37].position[0..8].ProcessValue.PosName := WSTRING#'';
   camDataBk[38].position[0..8].ProcessValue.PosName := WSTRING#'';
   camDataBk[39].position[0..8].ProcessValue.PosName := WSTRING#'';
   camDataBk[40].position[0..8].ProcessValue.PosName := WSTRING#'';
   camDataBk[41].position[0..8].ProcessValue.PosName := WSTRING#'';
   BA010.commands.Communication_Reset := FALSE;
   BA010.monitoring.error := FALSE;
   BA010.monitoring.status := 16#0000;
   BA010.configuration.disableAlarms := FALSE;
   BA010.configuration.SEND.connectionId := 16#0000;
   BA010.configuration.SEND.rid := 16#0000_0000;
   BA010.configuration.SEND.len := 16#0000;
   BA010.configuration.RCV.connectionId := 16#0000;
   BA010.configuration.RCV.rid := 16#0000_0000;
   BA015.commands.Communication_Reset := FALSE;
   BA015.monitoring.error := FALSE;
   BA015.monitoring.status := 16#0000;
   BA015.configuration.disableAlarms := FALSE;
   BA015.configuration.SEND.connectionId := 16#0000;
   BA015.configuration.SEND.rid := 16#0000_0000;
   BA015.configuration.SEND.len := 16#0000;
   BA015.configuration.RCV.connectionId := 16#0000;
   BA015.configuration.RCV.rid := 16#0000_0000;
   BA060.commands.Communication_Reset := FALSE;
   BA060.monitoring.error := FALSE;
   BA060.monitoring.status := 16#0000;
   BA060.configuration.disableAlarms := FALSE;
   BA060.configuration.SEND.connectionId := 16#0000;
   BA060.configuration.SEND.rid := 16#0000_0000;
   BA060.configuration.SEND.len := 16#0000;
   BA060.configuration.RCV.connectionId := 16#0000;
   BA060.configuration.RCV.rid := 16#0000_0000;
   BA040.commands.Communication_Reset := FALSE;
   BA040.monitoring.error := FALSE;
   BA040.monitoring.status := 16#0000;
   BA040.configuration.disableAlarms := FALSE;
   BA040.configuration.SEND.connectionId := 16#0000;
   BA040.configuration.SEND.rid := 16#0000_0000;
   BA040.configuration.SEND.len := 16#0000;
   BA040.configuration.RCV.connectionId := 16#0000;
   BA040.configuration.RCV.rid := 16#0000_0000;
   cmFFU.commands.Reset := FALSE;
   cmFFU.commands.Save := FALSE;
   cmFFU.monitoring.RPM_PV := 1250;
   cmFFU.monitoring.Alarm[0] := FALSE;
   cmFFU.monitoring.Alarm[1] := TRUE;
   cmFFU.monitoring.Alarm[2..6] := FALSE;
   cmFFU.monitoring.Error := FALSE;
   cmFFU.configuration.referenceDesignator := WSTRING#'cmFFU_LIU117';
   cmFFU.configuration.MB_Comm_Load.REQ := FALSE;
   cmFFU.configuration.MB_Comm_Load.PORT := 0;
   cmFFU.configuration.MB_Comm_Load.BAUD := 0;
   cmFFU.configuration.MB_Comm_Load.MB_DB.S_PORT := 16#FFFF;
   cmFFU.configuration.MB_Comm_Load.MB_DB.S_RESP_TO := 16#0000;
   cmFFU.configuration.MB_Comm_Load.MB_DB.S_ICHAR_GAP := 16#0000;
   cmFFU.configuration.MB_Comm_Load.MB_DB.S_RETRIES := 16#0000;
   cmFFU.configuration.MB_Comm_Load.MB_DB.S_MB_CRC := 16#00;
   cmFFU.configuration.MB_Comm_Load.PARITY := 0;
   cmFFU.configuration.MB_Comm_Load.DONE := FALSE;
   cmFFU.configuration.MB_Comm_Load.ERROR := FALSE;
   cmFFU.configuration.MB_Comm_Load.STATUS := 16#0000;
   cmFFU.configuration.MB_Master.REQ := FALSE;
   cmFFU.configuration.MB_Master.MB_ADDR := 0;
   cmFFU.configuration.MB_Master.MODE := 0;
   cmFFU.configuration.MB_Master.DATA_ADDR := 0;
   cmFFU.configuration.MB_Master.DATA_LEN := 0;
   cmFFU.configuration.MB_Master.DONE := FALSE;
   cmFFU.configuration.MB_Master.BUSY := FALSE;
   cmFFU.configuration.MB_Master.ERROR := FALSE;
   cmFFU.configuration.MB_Master.STATUS := 16#0000;
   cmFFU.configuration.MB_Master.DataPTR[1..2] := 0;
   cmFFU.configuration.RPM_SV := 0;
   DriveDiagConfig.driveObjects[0].referenceDesignator := WSTRING#'BA030AZSDR1';
   DriveDiagConfig.driveObjects[1].referenceDesignator := WSTRING#'BA030AZSDR2';
   DriveDiagConfig.driveObjects[2].referenceDesignator := WSTRING#'BA030AZSDR3';
   DriveDiagConfig.driveObjects[3].referenceDesignator := WSTRING#'';
   DriveDiagConfig.driveObjects[4].referenceDesignator := WSTRING#'BA030AZSDR5';
   DriveDiagConfig.driveObjects[5].referenceDesignator := WSTRING#'BA030AZSDR6';
   DriveDiagConfig.driveObjects[6].referenceDesignator := WSTRING#'BA030AZSDR7';
   DriveDiagConfig.driveObjects[7].referenceDesignator := WSTRING#'BA030AZSDR8';
   DriveDiagConfig.driveObjects[8].referenceDesignator := WSTRING#'BA030AZSDR9';
   DriveDiagConfig.driveObjects[9].referenceDesignator := WSTRING#'BA030AZSDR10';
   DriveDiagConfig.driveObjects[10].referenceDesignator := WSTRING#'BA030AZSDR11';
   DriveDiagConfig.driveObjects[11].referenceDesignator := WSTRING#'BA030AZSDR12';
   DriveDiagConfig.driveObjects[12].referenceDesignator := WSTRING#'BA030AZSDR13';
   DriveDiagConfig.driveObjects[13].referenceDesignator := WSTRING#'BA030AZSDR14';
   DriveDiagConfig.driveObjects[14].referenceDesignator := WSTRING#'BA030AZSDR15';
   DriveDiagConfig.driveObjects[15].referenceDesignator := WSTRING#'BA030AZSDR16';
   DriveDiagConfig.driveObjects[16].referenceDesignator := WSTRING#'BA030AZSDR17';
   DriveDiagConfig.driveObjects[17].referenceDesignator := WSTRING#'BA030AZSDR18';
   DriveDiagConfig.driveObjects[18].referenceDesignator := WSTRING#'BA030AZSDR19';
   DriveDiagConfig.driveObjects[19].referenceDesignator := WSTRING#'BA030AZSDR20';
   DriveDiagConfig.driveObjects[20].referenceDesignator := WSTRING#'BA030AZSDR21';
   DriveDiagConfig.driveObjects[21].referenceDesignator := WSTRING#'BA030AZSDR22';
   DriveDiagConfig.driveObjects[22].referenceDesignator := WSTRING#'BA030AZSDR23';
   DriveDiagConfig.driveObjects[23].referenceDesignator := WSTRING#'BA030AZSDR24';
   DriveDiagConfig.driveObjects[24].referenceDesignator := WSTRING#'BA030AZSDR25';
   DriveDiagConfig.driveObjects[25].referenceDesignator := WSTRING#'BA030AZSDR26';
   DriveDiagConfig.driveObjects[26].referenceDesignator := WSTRING#'BA030AZSDR27';
   DriveDiagConfig.driveObjects[27].referenceDesignator := WSTRING#'BA030AZSDR28';
   DriveDiagConfig.driveObjects[28].referenceDesignator := WSTRING#'BA030AZSDR29';
   DriveDiagConfig.driveObjects[29].referenceDesignator := WSTRING#'BA030AZSDR30';
   DriveDiagConfig.driveObjects[30].referenceDesignator := WSTRING#'BA030AZSDR31';
   DriveDiagConfig.driveObjects[31].referenceDesignator := WSTRING#'BA030AZSDR32';
   DriveDiagConfig.driveObjects[32].referenceDesignator := WSTRING#'BA030AZSDR33';
   DriveDiagConfig.driveObjects[33].referenceDesignator := WSTRING#'BA030AZSDR34';
   DriveDiagConfig.driveObjects[34].referenceDesignator := WSTRING#'BA030AZSDR35';
   DriveDiagConfig.driveObjects[35].referenceDesignator := WSTRING#'BA030AZSDR36';
   DriveDiagConfig.driveObjects[36].referenceDesignator := WSTRING#'BA030AZSDR37';
   DriveDiagConfig.driveObjects[37].referenceDesignator := WSTRING#'BA030AZSDR38';
   DriveDiagConfig.driveObjects[38].referenceDesignator := WSTRING#'BA030AZSDR39';
   DriveDiagConfig.driveObjects[39].referenceDesignator := WSTRING#'BA030AZSDR40';
   DriveDiagConfig.driveObjects[40].referenceDesignator := WSTRING#'BA030AZSDR41';
   DriveDiagConfig.driveObjects[41].referenceDesignator := WSTRING#'';
   DriveDiagConfig.driveObjects[0].axisDB := 263;
   DriveDiagConfig.driveObjects[1].axisDB := 141;
   DriveDiagConfig.driveObjects[2].axisDB := 143;
   DriveDiagConfig.driveObjects[3].axisDB := 0;
   DriveDiagConfig.driveObjects[4].axisDB := 144;
   DriveDiagConfig.driveObjects[5].axisDB := 145;
   DriveDiagConfig.driveObjects[6].axisDB := 146;
   DriveDiagConfig.driveObjects[7].axisDB := 147;
   DriveDiagConfig.driveObjects[8].axisDB := 152;
   DriveDiagConfig.driveObjects[9].axisDB := 151;
   DriveDiagConfig.driveObjects[10].axisDB := 148;
   DriveDiagConfig.driveObjects[11].axisDB := 149;
   DriveDiagConfig.driveObjects[12].axisDB := 153;
   DriveDiagConfig.driveObjects[13].axisDB := 150;
   DriveDiagConfig.driveObjects[14].axisDB := 154;
   DriveDiagConfig.driveObjects[15].axisDB := 155;
   DriveDiagConfig.driveObjects[16].axisDB := 156;
   DriveDiagConfig.driveObjects[17].axisDB := 157;
   DriveDiagConfig.driveObjects[18].axisDB := 158;
   DriveDiagConfig.driveObjects[19].axisDB := 159;
   DriveDiagConfig.driveObjects[20].axisDB := 171;
   DriveDiagConfig.driveObjects[21].axisDB := 172;
   DriveDiagConfig.driveObjects[22].axisDB := 163;
   DriveDiagConfig.driveObjects[23].axisDB := 162;
   DriveDiagConfig.driveObjects[24].axisDB := 167;
   DriveDiagConfig.driveObjects[25].axisDB := 166;
   DriveDiagConfig.driveObjects[26].axisDB := 161;
   DriveDiagConfig.driveObjects[27].axisDB := 160;
   DriveDiagConfig.driveObjects[28].axisDB := 165;
   DriveDiagConfig.driveObjects[29].axisDB := 164;
   DriveDiagConfig.driveObjects[30].axisDB := 168;
   DriveDiagConfig.driveObjects[31].axisDB := 169;
   DriveDiagConfig.driveObjects[32].axisDB := 170;
   DriveDiagConfig.driveObjects[33].axisDB := 177;
   DriveDiagConfig.driveObjects[34].axisDB := 175;
   DriveDiagConfig.driveObjects[35].axisDB := 178;
   DriveDiagConfig.driveObjects[36].axisDB := 173;
   DriveDiagConfig.driveObjects[37].axisDB := 174;
   DriveDiagConfig.driveObjects[38].axisDB := 180;
   DriveDiagConfig.driveObjects[39].axisDB := 179;
   DriveDiagConfig.driveObjects[40].axisDB := 176;
   DriveDiagConfig.driveObjects[41].axisDB := 0;
   DriveDiagConfig.driveObjects[0..2].sinaType := 124;
   DriveDiagConfig.driveObjects[3].sinaType := 0;
   DriveDiagConfig.driveObjects[4..40].sinaType := 124;
   DriveDiagConfig.driveObjects[41].sinaType := 0;
   DriveDiagConfig.driveObjects[0].sinaHwID := 259;
   DriveDiagConfig.driveObjects[1].sinaHwID := 517;
   DriveDiagConfig.driveObjects[2].sinaHwID := 818;
   DriveDiagConfig.driveObjects[3].sinaHwID := 0;
   DriveDiagConfig.driveObjects[4].sinaHwID := 519;
   DriveDiagConfig.driveObjects[5].sinaHwID := 523;
   DriveDiagConfig.driveObjects[6].sinaHwID := 527;
   DriveDiagConfig.driveObjects[7].sinaHwID := 529;
   DriveDiagConfig.driveObjects[8].sinaHwID := 541;
   DriveDiagConfig.driveObjects[9].sinaHwID := 547;
   DriveDiagConfig.driveObjects[10].sinaHwID := 559;
   DriveDiagConfig.driveObjects[11].sinaHwID := 561;
   DriveDiagConfig.driveObjects[12].sinaHwID := 564;
   DriveDiagConfig.driveObjects[13].sinaHwID := 569;
   DriveDiagConfig.driveObjects[14].sinaHwID := 568;
   DriveDiagConfig.driveObjects[15].sinaHwID := 571;
   DriveDiagConfig.driveObjects[16].sinaHwID := 573;
   DriveDiagConfig.driveObjects[17].sinaHwID := 577;
   DriveDiagConfig.driveObjects[18].sinaHwID := 659;
   DriveDiagConfig.driveObjects[19].sinaHwID := 660;
   DriveDiagConfig.driveObjects[20].sinaHwID := 589;
   DriveDiagConfig.driveObjects[21].sinaHwID := 596;
   DriveDiagConfig.driveObjects[22].sinaHwID := 654;
   DriveDiagConfig.driveObjects[23].sinaHwID := 667;
   DriveDiagConfig.driveObjects[24].sinaHwID := 671;
   DriveDiagConfig.driveObjects[25].sinaHwID := 682;
   DriveDiagConfig.driveObjects[26].sinaHwID := 620;
   DriveDiagConfig.driveObjects[27].sinaHwID := 626;
   DriveDiagConfig.driveObjects[28].sinaHwID := 684;
   DriveDiagConfig.driveObjects[29].sinaHwID := 686;
   DriveDiagConfig.driveObjects[30].sinaHwID := 605;
   DriveDiagConfig.driveObjects[31].sinaHwID := 635;
   DriveDiagConfig.driveObjects[32].sinaHwID := 663;
   DriveDiagConfig.driveObjects[33].sinaHwID := 690;
   DriveDiagConfig.driveObjects[34].sinaHwID := 649;
   DriveDiagConfig.driveObjects[35].sinaHwID := 692;
   DriveDiagConfig.driveObjects[36].sinaHwID := 657;
   DriveDiagConfig.driveObjects[37].sinaHwID := 697;
   DriveDiagConfig.driveObjects[38].sinaHwID := 665;
   DriveDiagConfig.driveObjects[39].sinaHwID := 666;
   DriveDiagConfig.driveObjects[40].sinaHwID := 653;
   DriveDiagConfig.driveObjects[41].sinaHwID := 0;
   DriveDiagConfig.driveObjects[0..1].sinaDriveObjectNo := 3;
   DriveDiagConfig.driveObjects[2].sinaDriveObjectNo := 4;
   DriveDiagConfig.driveObjects[3].sinaDriveObjectNo := 1;
   DriveDiagConfig.driveObjects[4].sinaDriveObjectNo := 2;
   DriveDiagConfig.driveObjects[5].sinaDriveObjectNo := 3;
   DriveDiagConfig.driveObjects[6].sinaDriveObjectNo := 4;
   DriveDiagConfig.driveObjects[7].sinaDriveObjectNo := 10;
   DriveDiagConfig.driveObjects[8].sinaDriveObjectNo := 5;
   DriveDiagConfig.driveObjects[9..10].sinaDriveObjectNo := 6;
   DriveDiagConfig.driveObjects[11].sinaDriveObjectNo := 2;
   DriveDiagConfig.driveObjects[12].sinaDriveObjectNo := 3;
   DriveDiagConfig.driveObjects[13].sinaDriveObjectNo := 4;
   DriveDiagConfig.driveObjects[14..40].sinaDriveObjectNo := 5;
   DriveDiagConfig.driveObjects[41].sinaDriveObjectNo := 1;
   DriveDiagInterfaceHmi.diagStatus.hmi.referenceDesignator := WSTRING#'';
   DriveDiagInterfaceHmi.diagStatus.hmi.driveIndex := 0;
   DriveDiagInterfaceHmi.diagStatus.hmi.axisStatusScreenActive := FALSE;
   DriveDiagInterfaceHmi.diagStatus.hmi.sinaStatusScreenActive := FALSE;
   DriveDiagInterfaceHmi.diagStatus.hmi.sinaAlarmScreenActive := FALSE;
   DriveDiagInterfaceHmi.diagStatus.hmi.sinaEposScreenActive := FALSE;
   DriveDiagInterfaceHmi.diagStatus.hmi.sinaSafetyScreenActive := FALSE;
   DriveDiagInterfaceHmi.diagStatus.axis."type" := 0;
   DriveDiagInterfaceHmi.diagStatus.axis.values.position := 0.0;
   DriveDiagInterfaceHmi.diagStatus.axis.values.velocity := 0.0;
   DriveDiagInterfaceHmi.diagStatus.axis.values.actualPosition := 0.0;
   DriveDiagInterfaceHmi.diagStatus.axis.values.actualVelocity := 0.0;
   DriveDiagInterfaceHmi.diagStatus.axis.values.actualSpeed := 0.0;
   DriveDiagInterfaceHmi.diagStatus.axis.statusAxis.statusWord := 16#0000_0000;
   DriveDiagInterfaceHmi.diagStatus.axis.statusAxis.statusWord2 := 16#0000_0000;
   DriveDiagInterfaceHmi.diagStatus.axis.statusAxis.warningWord := 16#0000_0000;
   DriveDiagInterfaceHmi.diagStatus.axis.statusAxis.errorWord := 16#0000_0000;
   DriveDiagInterfaceHmi.diagStatus.axis.statusAxis.status.bit00_Enable := FALSE;
   DriveDiagInterfaceHmi.diagStatus.axis.statusAxis.status.bit01_Error := FALSE;
   DriveDiagInterfaceHmi.diagStatus.axis.statusAxis.status.bit02_RestartActive := FALSE;
   DriveDiagInterfaceHmi.diagStatus.axis.statusAxis.status.bit03_OnlineStartValuesChanged := FALSE;
   DriveDiagInterfaceHmi.diagStatus.axis.statusAxis.status.bit04_ControlPanelActive := FALSE;
   DriveDiagInterfaceHmi.diagStatus.axis.statusAxis.status.bit05_HomingDone := FALSE;
   DriveDiagInterfaceHmi.diagStatus.axis.statusAxis.status.bit06_Done := FALSE;
   DriveDiagInterfaceHmi.diagStatus.axis.statusAxis.status.bit07_Standstill := FALSE;
   DriveDiagInterfaceHmi.diagStatus.axis.statusAxis.status.bit08_PositioningCommand := FALSE;
   DriveDiagInterfaceHmi.diagStatus.axis.statusAxis.status.bit09_JogCommand := FALSE;
   DriveDiagInterfaceHmi.diagStatus.axis.statusAxis.status.bit10_VelocityCommand := FALSE;
   DriveDiagInterfaceHmi.diagStatus.axis.statusAxis.status.bit11_HomingCommand := FALSE;
   DriveDiagInterfaceHmi.diagStatus.axis.statusAxis.status.bit12_ConstantVelocity := FALSE;
   DriveDiagInterfaceHmi.diagStatus.axis.statusAxis.status.bit13_Accelerating := FALSE;
   DriveDiagInterfaceHmi.diagStatus.axis.statusAxis.status.bit14_Decelerating := FALSE;
   DriveDiagInterfaceHmi.diagStatus.axis.statusAxis.status.bit15_SWLimitMinActive := FALSE;
   DriveDiagInterfaceHmi.diagStatus.axis.statusAxis.status.bit16_SWLimitMaxActive := FALSE;
   DriveDiagInterfaceHmi.diagStatus.axis.statusAxis.status.bit17_HWLimitMinActive := FALSE;
   DriveDiagInterfaceHmi.diagStatus.axis.statusAxis.status.bit18_HWLimitMaxActive := FALSE;
   DriveDiagInterfaceHmi.diagStatus.axis.statusAxis.status.bit19_Reserved := FALSE;
   DriveDiagInterfaceHmi.diagStatus.axis.statusAxis.status.bit20_Reserved := FALSE;
   DriveDiagInterfaceHmi.diagStatus.axis.statusAxis.status.bit21_Synchronizing := FALSE;
   DriveDiagInterfaceHmi.diagStatus.axis.statusAxis.status.bit22_Synchronous := FALSE;
   DriveDiagInterfaceHmi.diagStatus.axis.statusAxis.status.bit23_SuperimposedMotionCommand := FALSE;
   DriveDiagInterfaceHmi.diagStatus.axis.statusAxis.status.bit24_PhasingCommand := FALSE;
   DriveDiagInterfaceHmi.diagStatus.axis.statusAxis.status.bit25_AxisSimulation := FALSE;
   DriveDiagInterfaceHmi.diagStatus.axis.statusAxis.status.bit26_TorqueLimitingCommand := FALSE;
   DriveDiagInterfaceHmi.diagStatus.axis.statusAxis.status.bit27_InLimitation := FALSE;
   DriveDiagInterfaceHmi.diagStatus.axis.statusAxis.status.bit28_NonPositionControlled := FALSE;
   DriveDiagInterfaceHmi.diagStatus.axis.statusAxis.status.bit29_KinematicsMotionCommand := FALSE;
   DriveDiagInterfaceHmi.diagStatus.axis.statusAxis.status.bit30_InClamping := FALSE;
   DriveDiagInterfaceHmi.diagStatus.axis.statusAxis.status.bit31_MotionInCommand := FALSE;
   DriveDiagInterfaceHmi.diagStatus.axis.statusAxis.status2.bit00_StopCommand := FALSE;
   DriveDiagInterfaceHmi.diagStatus.axis.statusAxis.status2.bit01_DesynchronizingCommand := FALSE;
   DriveDiagInterfaceHmi.diagStatus.axis.statusAxis.status2.bit02_PassingBacklash := FALSE;
   DriveDiagInterfaceHmi.diagStatus.axis.statusAxis.status2.bit03_PhasingCommandWaiting := FALSE;
   DriveDiagInterfaceHmi.diagStatus.axis.statusAxis.status2.bit04_OffsetCommand := FALSE;
   DriveDiagInterfaceHmi.diagStatus.axis.statusAxis.status2.bit05_OffsetCommandWaiting := FALSE;
   DriveDiagInterfaceHmi.diagStatus.axis.statusAxis.status2.bit06_MotionInSuperimposedCommand := FALSE;
   DriveDiagInterfaceHmi.diagStatus.axis.statusAxis.status2.bit07_HaltSuperimposedCommand := FALSE;
   DriveDiagInterfaceHmi.diagStatus.axis.statusAxis.status2.bit08_Reserved := FALSE;
   DriveDiagInterfaceHmi.diagStatus.axis.statusAxis.status2.bit09_Reserved := FALSE;
   DriveDiagInterfaceHmi.diagStatus.axis.statusAxis.status2.bit10_Reserved := FALSE;
   DriveDiagInterfaceHmi.diagStatus.axis.statusAxis.status2.bit11_Reserved := FALSE;
   DriveDiagInterfaceHmi.diagStatus.axis.statusAxis.status2.bit12_Reserved := FALSE;
   DriveDiagInterfaceHmi.diagStatus.axis.statusAxis.status2.bit13_Reserved := FALSE;
   DriveDiagInterfaceHmi.diagStatus.axis.statusAxis.status2.bit14_Reserved := FALSE;
   DriveDiagInterfaceHmi.diagStatus.axis.statusAxis.status2.bit15_Reserved := FALSE;
   DriveDiagInterfaceHmi.diagStatus.axis.statusAxis.status2.bit16_Reserved := FALSE;
   DriveDiagInterfaceHmi.diagStatus.axis.statusAxis.status2.bit17_Reserved := FALSE;
   DriveDiagInterfaceHmi.diagStatus.axis.statusAxis.status2.bit18_Reserved := FALSE;
   DriveDiagInterfaceHmi.diagStatus.axis.statusAxis.status2.bit19_Reserved := FALSE;
   DriveDiagInterfaceHmi.diagStatus.axis.statusAxis.status2.bit20_Reserved := FALSE;
   DriveDiagInterfaceHmi.diagStatus.axis.statusAxis.status2.bit21_Reserved := FALSE;
   DriveDiagInterfaceHmi.diagStatus.axis.statusAxis.status2.bit22_Reserved := FALSE;
   DriveDiagInterfaceHmi.diagStatus.axis.statusAxis.status2.bit23_Reserved := FALSE;
   DriveDiagInterfaceHmi.diagStatus.axis.statusAxis.status2.bit24_Reserved := FALSE;
   DriveDiagInterfaceHmi.diagStatus.axis.statusAxis.status2.bit25_Reserved := FALSE;
   DriveDiagInterfaceHmi.diagStatus.axis.statusAxis.status2.bit26_Reserved := FALSE;
   DriveDiagInterfaceHmi.diagStatus.axis.statusAxis.status2.bit27_Reserved := FALSE;
   DriveDiagInterfaceHmi.diagStatus.axis.statusAxis.status2.bit28_Reserved := FALSE;
   DriveDiagInterfaceHmi.diagStatus.axis.statusAxis.status2.bit29_Reserved := FALSE;
   DriveDiagInterfaceHmi.diagStatus.axis.statusAxis.status2.bit30_Reserved := FALSE;
   DriveDiagInterfaceHmi.diagStatus.axis.statusAxis.status2.bit31_Reserved := FALSE;
   DriveDiagInterfaceHmi.diagStatus.axis.statusAxis.warning.bit00_SystemWarning := FALSE;
   DriveDiagInterfaceHmi.diagStatus.axis.statusAxis.warning.bit01_ConfigWarning := FALSE;
   DriveDiagInterfaceHmi.diagStatus.axis.statusAxis.warning.bit02_UserWarning := FALSE;
   DriveDiagInterfaceHmi.diagStatus.axis.statusAxis.warning.bit03_CommandNotAccepted := FALSE;
   DriveDiagInterfaceHmi.diagStatus.axis.statusAxis.warning.bit04_DriveWarning := FALSE;
   DriveDiagInterfaceHmi.diagStatus.axis.statusAxis.warning.bit05_SensorWarning := FALSE;
   DriveDiagInterfaceHmi.diagStatus.axis.statusAxis.warning.bit06_DynamicWarning := FALSE;
   DriveDiagInterfaceHmi.diagStatus.axis.statusAxis.warning.bit07_CommunicationWarning := FALSE;
   DriveDiagInterfaceHmi.diagStatus.axis.statusAxis.warning.bit08_SWLimitMin := FALSE;
   DriveDiagInterfaceHmi.diagStatus.axis.statusAxis.warning.bit09_SWLimitMax := FALSE;
   DriveDiagInterfaceHmi.diagStatus.axis.statusAxis.warning.bit10_HomingWarning := FALSE;
   DriveDiagInterfaceHmi.diagStatus.axis.statusAxis.warning.bit11_FollowingErrorWarning := FALSE;
   DriveDiagInterfaceHmi.diagStatus.axis.statusAxis.warning.bit12_PositioningWarning := FALSE;
   DriveDiagInterfaceHmi.diagStatus.axis.statusAxis.warning.bit13_PeripheralWarning := FALSE;
   DriveDiagInterfaceHmi.diagStatus.axis.statusAxis.warning.bit14_SynchronousWarning := FALSE;
   DriveDiagInterfaceHmi.diagStatus.axis.statusAxis.warning.bit15_AdaptionWarning := FALSE;
   DriveDiagInterfaceHmi.diagStatus.axis.statusAxis.warning.bit16_Reserved := FALSE;
   DriveDiagInterfaceHmi.diagStatus.axis.statusAxis.warning.bit17_Reserved := FALSE;
   DriveDiagInterfaceHmi.diagStatus.axis.statusAxis.warning.bit18_Reserved := FALSE;
   DriveDiagInterfaceHmi.diagStatus.axis.statusAxis.warning.bit19_Reserved := FALSE;
   DriveDiagInterfaceHmi.diagStatus.axis.statusAxis.warning.bit20_Reserved := FALSE;
   DriveDiagInterfaceHmi.diagStatus.axis.statusAxis.warning.bit21_Reserved := FALSE;
   DriveDiagInterfaceHmi.diagStatus.axis.statusAxis.warning.bit22_Reserved := FALSE;
   DriveDiagInterfaceHmi.diagStatus.axis.statusAxis.warning.bit23_Reserved := FALSE;
   DriveDiagInterfaceHmi.diagStatus.axis.statusAxis.warning.bit24_Reserved := FALSE;
   DriveDiagInterfaceHmi.diagStatus.axis.statusAxis.warning.bit25_Reserved := FALSE;
   DriveDiagInterfaceHmi.diagStatus.axis.statusAxis.warning.bit26_Reserved := FALSE;
   DriveDiagInterfaceHmi.diagStatus.axis.statusAxis.warning.bit27_Reserved := FALSE;
   DriveDiagInterfaceHmi.diagStatus.axis.statusAxis.warning.bit28_Reserved := FALSE;
   DriveDiagInterfaceHmi.diagStatus.axis.statusAxis.warning.bit29_Reserved := FALSE;
   DriveDiagInterfaceHmi.diagStatus.axis.statusAxis.warning.bit30_Reserved := FALSE;
   DriveDiagInterfaceHmi.diagStatus.axis.statusAxis.warning.bit31_Reserved := FALSE;
   DriveDiagInterfaceHmi.diagStatus.axis.statusAxis.error.bit00_SystemFault := FALSE;
   DriveDiagInterfaceHmi.diagStatus.axis.statusAxis.error.bit01_ConfigFault := FALSE;
   DriveDiagInterfaceHmi.diagStatus.axis.statusAxis.error.bit02_UserFault := FALSE;
   DriveDiagInterfaceHmi.diagStatus.axis.statusAxis.error.bit03_CommandNotAccepted := FALSE;
   DriveDiagInterfaceHmi.diagStatus.axis.statusAxis.error.bit04_DriveFault := FALSE;
   DriveDiagInterfaceHmi.diagStatus.axis.statusAxis.error.bit05_SensorFault := FALSE;
   DriveDiagInterfaceHmi.diagStatus.axis.statusAxis.error.bit06_DynamicError := FALSE;
   DriveDiagInterfaceHmi.diagStatus.axis.statusAxis.error.bit07_CommunicationFault := FALSE;
   DriveDiagInterfaceHmi.diagStatus.axis.statusAxis.error.bit08_SWLimit := FALSE;
   DriveDiagInterfaceHmi.diagStatus.axis.statusAxis.error.bit09_HWLimit := FALSE;
   DriveDiagInterfaceHmi.diagStatus.axis.statusAxis.error.bit10_HomingError := FALSE;
   DriveDiagInterfaceHmi.diagStatus.axis.statusAxis.error.bit11_FollowingErrorFault := FALSE;
   DriveDiagInterfaceHmi.diagStatus.axis.statusAxis.error.bit12_PositioningFault := FALSE;
   DriveDiagInterfaceHmi.diagStatus.axis.statusAxis.error.bit13_PeripheralError := FALSE;
   DriveDiagInterfaceHmi.diagStatus.axis.statusAxis.error.bit14_SynchronousError := FALSE;
   DriveDiagInterfaceHmi.diagStatus.axis.statusAxis.error.bit15_AdaptionError := FALSE;
   DriveDiagInterfaceHmi.diagStatus.axis.statusAxis.error.bit16_Reserved := FALSE;
   DriveDiagInterfaceHmi.diagStatus.axis.statusAxis.error.bit17_Reserved := FALSE;
   DriveDiagInterfaceHmi.diagStatus.axis.statusAxis.error.bit18_Reserved := FALSE;
   DriveDiagInterfaceHmi.diagStatus.axis.statusAxis.error.bit19_Reserved := FALSE;
   DriveDiagInterfaceHmi.diagStatus.axis.statusAxis.error.bit20_Reserved := FALSE;
   DriveDiagInterfaceHmi.diagStatus.axis.statusAxis.error.bit21_Reserved := FALSE;
   DriveDiagInterfaceHmi.diagStatus.axis.statusAxis.error.bit22_Reserved := FALSE;
   DriveDiagInterfaceHmi.diagStatus.axis.statusAxis.error.bit23_Reserved := FALSE;
   DriveDiagInterfaceHmi.diagStatus.axis.statusAxis.error.bit24_Reserved := FALSE;
   DriveDiagInterfaceHmi.diagStatus.axis.statusAxis.error.bit25_Reserved := FALSE;
   DriveDiagInterfaceHmi.diagStatus.axis.statusAxis.error.bit26_Reserved := FALSE;
   DriveDiagInterfaceHmi.diagStatus.axis.statusAxis.error.bit27_Reserved := FALSE;
   DriveDiagInterfaceHmi.diagStatus.axis.statusAxis.error.bit28_Reserved := FALSE;
   DriveDiagInterfaceHmi.diagStatus.axis.statusAxis.error.bit29_Reserved := FALSE;
   DriveDiagInterfaceHmi.diagStatus.axis.statusAxis.error.bit30_Reserved := FALSE;
   DriveDiagInterfaceHmi.diagStatus.axis.statusAxis.error.bit31_Reserved := FALSE;
   DriveDiagInterfaceHmi.diagStatus.axis.statusAxis.errorDetail.number := 0;
   DriveDiagInterfaceHmi.diagStatus.axis.statusAxis.errorDetail.reaction := 0;
   DriveDiagInterfaceHmi.diagStatus.axis.statusSensor.operativeSensor := 1;
   DriveDiagInterfaceHmi.diagStatus.axis.statusSensor.sensor[1..4].state := 0;
   DriveDiagInterfaceHmi.diagStatus.axis.statusSensor.sensor[1..4].communicationOK := FALSE;
   DriveDiagInterfaceHmi.diagStatus.axis.statusSensor.sensor[1..4].error := FALSE;
   DriveDiagInterfaceHmi.diagStatus.axis.statusSensor.sensor[1..4].control := FALSE;
   DriveDiagInterfaceHmi.diagStatus.axis.statusSensor.sensor[1..4].position := 0.0;
   DriveDiagInterfaceHmi.diagStatus.axis.statusSensor.sensor[1..4].velocity := 0.0;
   DriveDiagInterfaceHmi.diagStatus.axis.statusSensor.sensor[1..4].adaptionState := 0;
   DriveDiagInterfaceHmi.diagStatus.axis.statusSensor.sensor[1..4].adjusted := 0;
   DriveDiagInterfaceHmi.diagStatus.axis.statusPositioning.targetPosition := 0.0;
   DriveDiagInterfaceHmi.diagStatus.axis.statusPositioning.followingError := 0.0;
   DriveDiagInterfaceHmi.diagStatus.axis.units.lengthUnit := 0;
   DriveDiagInterfaceHmi.diagStatus.axis.units.velocityUnit := 0;
   DriveDiagInterfaceHmi.diagStatus.sina.sinaType := 0;
   DriveDiagInterfaceHmi.diagStatus.sina.controlWord := 16#0000;
   DriveDiagInterfaceHmi.diagStatus.sina.statusWord := 16#0000;
   DriveDiagInterfaceHmi.diagStatus.sina.telegramNo := 0;
   DriveDiagInterfaceHmi.diagStatus.sina.eposStatusWord1 := 16#0000;
   DriveDiagInterfaceHmi.diagStatus.sina.eposStatusWord2 := 16#0000;
   DriveDiagInterfaceHmi.diagStatus.sina.operatingDisplay := 0;
   DriveDiagInterfaceHmi.diagStatus.sina.override := 0.0;
   DriveDiagInterfaceHmi.diagStatus.sina.posSetValue := 0.0;
   DriveDiagInterfaceHmi.diagStatus.sina.posActValue := 0.0;
   DriveDiagInterfaceHmi.diagStatus.sina.velSetValue := 0.0;
   DriveDiagInterfaceHmi.diagStatus.sina.velActValue := 0.0;
   DriveDiagInterfaceHmi.diagStatus.sina.lengthUnit := 0;
   DriveDiagInterfaceHmi.diagStatus.sina.velocityUnit := 0;
   DriveDiagInterfaceHmi.diagStatus.sina.residualDistance := 0.0;
   DriveDiagInterfaceHmi.diagStatus.sina.followingError := 0.0;
   DriveDiagInterfaceHmi.diagStatus.sina.posControlWord := 16#0000;
   DriveDiagInterfaceHmi.diagStatus.sina.posStatusWord := 16#0000;
   DriveDiagInterfaceHmi.diagStatus.sina.blockSelected := 0;
   DriveDiagInterfaceHmi.diagStatus.sina.blockActive := 0;
   DriveDiagInterfaceHmi.diagStatus.sina.mdiPosSetValue := 0.0;
   DriveDiagInterfaceHmi.diagStatus.sina.faultCode[0..7] := 16#0000;
   DriveDiagInterfaceHmi.diagStatus.sina.alarmCode[0..3] := 16#0000;
   DriveDiagInterfaceHmi.diagStatus.sina.speedSetValue := 0.0;
   DriveDiagInterfaceHmi.diagStatus.sina.speedActValue := 0.0;
   DriveDiagInterfaceHmi.diagStatus.sina.safetyStatusWord := 16#0000;
END_DATA_BLOCK
